FUNCTION_BLOCK FB_Mover EXTENDS CyclicBase IMPLEMENTS IMover, IDynamics
VAR
	axesEnable		: AxisPower(_axis);
	axesReset		: AxesReset(_axis);
	axesMoveTo 		: MoveMoverToPosition(_axis) := (Gap := 100.0);
	axesHalt 		: HaltMover(_axis);
	axesReadError : Tc2_MC2.MC_ReadAxisError;
	_axis 			: AXIS_REF;
	_identInGroup : INT;
	_trackLength : MC_LREAL;
	_targetPos : LREAL;
	_MoverErrorId : DWORD;
	_arrZones : ARRAY[1..4] OF DINT;
	_arrVelocities : ARRAY[1..4] OF mc_LREAL;
END_VAR

PROPERTY PUBLIC Acceleration : mc_lreal
GET
Acceleration := axesMoveTo.Acceleration;
END_GET
SET
axesMoveTo.Acceleration := Acceleration;
END_SET
END_PROPERTY

PROPERTY PUBLIC AxisRef : reference to AXIS_REF
GET
AxisRef REF= THIS^._axis;
END_GET
END_PROPERTY

METHOD PUBLIC  Cycle : BOOL
VAR_INPUT
END_VAR
axesMoveTo.Cycle();
axesHalt.Cycle();
axesReset.Cycle();
_axis.ReadStatus();
axesEnable.Cycle();
axesReadError(Axis := _axis, Enable := TRUE, AxisErrorID => _MoverErrorId);
END_METHOD

PROPERTY PUBLIC Deceleration : mc_lreal
GET
Deceleration := axesMoveTo.Deceleration;
END_GET
SET
axesMoveTo.Deceleration := Deceleration;
END_SET
END_PROPERTY

METHOD PUBLIC DisableAxis : BOOL
VAR_INPUT
END_VAR
DisableAxis := axesEnable.Disable();
END_METHOD

METHOD PUBLIC EnableAxis : BOOL
VAR_INPUT
END_VAR
EnableAxis := axesEnable.Enable();
END_METHOD

PROPERTY PUBLIC Gap : mc_lreal
GET
Gap := axesMoveTo.Gap;
END_GET
SET
axesMoveTo.Gap := Gap;
END_SET
END_PROPERTY

METHOD PUBLIC HaltAxis : BOOL
VAR_INPUT
END_VAR
IF NOT axesHalt.Busy THEN
	axesHalt.Execute();
	HaltAxis := TRUE;
	axesMoveTo.Abort();
END_IF
END_METHOD

METHOD PUBLIC HasCommand : BOOL
VAR_INPUT
END_VAR
HasCommand := axesMoveTo.Busy;
END_METHOD

METHOD hasError : BOOL
VAR_INPUT
END_VAR
hasError := _axis.Status.Error;
END_METHOD

PROPERTY PUBLIC IdentInGroup : int
GET
IdentInGroup := _identInGroup;
END_GET
SET
_identInGroup := IdentInGroup;
END_SET
END_PROPERTY

METHOD isAtPosition : BOOL
VAR_INPUT
	position : MC_LREAL;
END_VAR
IF position > 1 THEN
	IF _axis.NcToPlc.ModuloActPos < position + 1 AND _axis.NcToPlc.ModuloActPos > position - 1 THEN
		isAtPosition := TRUE;
	END_IF  
ELSE
	IF _axis.NcToPlc.ModuloActPos < position + 1 AND _axis.NcToPlc.ModuloActPos > 0.0  
		OR _axis.NcToPlc.ModuloActPos < _trackLength AND _axis.NcToPlc.ModuloActPos > _trackLength - 1 THEN
		isAtPosition := TRUE;
	END_IF
END_IF
END_METHOD

METHOD PUBLIC isDetected : BOOL
VAR_INPUT
END_VAR
IF _axis.NcToPlc.AxisId = 0 THEN
	RETURN;
END_IF
isDetected := true;
END_METHOD

METHOD isEnabled : BOOL
VAR_INPUT
END_VAR
isEnabled := not _axis.Status.Disabled;
END_METHOD

METHOD PUBLIC isPastPosition : BOOL
VAR_INPUT
	position : MC_LREAL;
END_VAR
IF position > 1 THEN
	IF _axis.NcToPlc.ModuloActPos > position THEN
		isPastPosition := TRUE;
	END_IF  
END_IF
END_METHOD

METHOD PUBLIC isStationary : BOOL
VAR_INPUT
END_VAR
isStationary := _axis.NcToPlc.SetVelo = 0;
END_METHOD

PROPERTY PUBLIC Jerk : mc_lreal
GET
Jerk := axesMoveTo.Jerk;
END_GET
SET
axesMoveTo.Jerk := Jerk;
END_SET
END_PROPERTY

METHOD PROTECTED ModuloToAbs : mc_lreal
VAR_INPUT
	moduloPositionDemand: MC_LREAL;
	_backwardsAllowed : BOOL;
END_VAR
//---------code to set actual position from modulo command----------------------
IF NOT _backwardsAllowed THEN
	//--------if you want to go forward-------------------------------------------------------------
	//---------if SetPos is greater than current actual then move to that position--------------------
	//---------else current position is greater, increase moduloturn count by 1 before set---------------
	IF moduloPositionDemand > _axis.NcToPlc.ModuloActPos THEN
		ModuloToAbs := (DINT_TO_LREAL(_Axis.NcToPlc.ModuloActTurns)*_trackLength) + moduloPositionDemand;
	ELSE
		ModuloToAbs := (DINT_TO_LREAL(_Axis.NcToPlc.ModuloActTurns + 1)*_trackLength) + moduloPositionDemand;
	END_IF
ELSE
	//--------if you want to go backwards--------------------------------
	//--------if setPos is less than current actual then move to that position---------------------
	//---------else current position is less, decrease moduloturn count by 1 before set------------
	IF moduloPositionDemand < _axis.NcToPlc.ModuloActPos THEN
		ModuloToAbs := (DINT_TO_LREAL(_Axis.NcToPlc.ModuloActTurns)*_trackLength) + moduloPositionDemand;
	ELSE
		ModuloToAbs := (DINT_TO_LREAL(_Axis.NcToPlc.ModuloActTurns-1)*_trackLength) + moduloPositionDemand;
	END_IF
END_IF
END_METHOD

PROPERTY MoverErrorId : dword
GET
MoverErrorId := _MoverErrorId;
END_GET
SET
_MoverErrorId := MoverErrorId;
END_SET
END_PROPERTY

METHOD PUBLIC MoveTo : BOOL
VAR_INPUT
	Position : MC_LREAL;
	Velocity : MC_LREAL;
	BackwardMove : BOOL;
END_VAR
IF NOT isAtPosition(position := Position) THEN
	IF NOT axesMoveTo.Busy THEN
		axesMoveTo.MoveTo(Position := ModuloToAbs(Position, BackwardMove), Velocity := Velocity);
		MoveTo := TRUE;
		_targetPos := Position;
	END_IF
END_IF
END_METHOD

METHOD PUBLIC ResetAxis : BOOL
VAR_INPUT
END_VAR
VAR
END_VAR
axesReset.Execute();
axesMoveTo.Abort();
axesHalt.Abort();
END_METHOD

PROPERTY PUBLIC TrackLength : MC_LREAL
GET
TrackLength := _trackLength;
END_GET
SET
_trackLength := TrackLength;
END_SET
END_PROPERTY

PROPERTY Zones : array[1..4] of dint
GET
Zones := _arrZones;
END_GET
SET
_arrZones := Zones;
END_SET
END_PROPERTY

PROPERTY ZoneVelocities : array[1..4] of mc_lreal
GET
ZoneVelocities := _arrVelocities;
END_GET
SET
_arrVelocities := ZoneVelocities;
END_SET
END_PROPERTY

END_FUNCTION_BLOCK

(* stored: Version 1.1.0.1, ProductVersion 3.1.4024.12
   POU FB_Mover: Id {8d73ea9c-992c-45cc-86ce-646b77b87654}, SpecialFunc None
   Folder Methods: Id {11c06f36-011b-43e0-ba96-46cd7b32bc9c}
   Folder Properties: Id {a74425e5-3b65-414c-b3c2-ebd17b6452b3}
   Property Acceleration: Id {189e8681-4788-4e2c-a142-1a297a08acd8}
   Get Get: Id {2a072cec-dc98-4e3e-832d-7b1661a2a48e}
   Set Set: Id {ac96b1c2-72ed-4693-b71f-9fbcd2a6afd7}
   Property AxisRef: Id {09529bdd-b0dc-4149-87fe-1e673dd7e409}
   Get Get: Id {8057bced-3b30-4db1-bed6-093c25080d45}
   Method Cycle: Id {df169178-ee0f-491e-a015-1bc9be6eb17c}
   Property Deceleration: Id {c85f3f81-4f88-4542-92dd-87b98693dee4}
   Get Get: Id {578458d3-d8f3-428d-9fc2-a6d51c86d4b3}
   Set Set: Id {b756c826-c655-4fcf-88a7-bb105c6d7b9b}
   Method DisableAxis: Id {c70711cc-2b37-46ae-851d-9b38023a0d20}
   Method EnableAxis: Id {b661d1e7-696c-4d63-afd0-3918405db14b}
   Property Gap: Id {e555cbf2-c13b-4254-9bb2-744e7edb7578}
   Get Get: Id {a0479bdd-653c-4687-93eb-073972457858}
   Set Set: Id {8af53078-5c57-4e61-9843-6d0cf8d12af4}
   Method HaltAxis: Id {fcdbac8a-7893-40e4-99e2-5063962a86e4}
   Method HasCommand: Id {87052920-e2d9-4076-9a13-adb664b2e231}
   Method hasError: Id {c0115f9f-d324-4748-af93-c56fdaaf010c}
   Property IdentInGroup: Id {ef5d4455-d34d-4ca1-b17f-13425cd154ed}
   Get Get: Id {de907afb-d6b6-48b4-8857-851ff7b7bba8}
   Set Set: Id {4b095c67-211b-468a-8be3-48d4ac28c572}
   Method isAtPosition: Id {2f15d1ba-ddfc-4b9e-afe4-5a0e456096bb}
   Method isDetected: Id {4d5c40c2-9705-45a9-9e7d-17e4126ba8ba}
   Method isEnabled: Id {5db97821-4f9e-4a12-8756-664c948ce8d4}
   Method isPastPosition: Id {9fa8306a-b12e-4f44-a97a-94fb24ba9f28}
   Method isStationary: Id {38624f60-08a0-42b1-ae6f-e7cfbf630206}
   Property Jerk: Id {08f26a51-2cac-4172-adfd-333cdfa23de5}
   Get Get: Id {b3f4bc4a-fc36-46a7-a0ff-605d9a2ddc0b}
   Set Set: Id {e967ae27-5c59-444d-a01e-9a7980e3667f}
   Method ModuloToAbs: Id {3e98c8eb-3ddf-4e09-8a71-47cbd2f60d1c}
   Property MoverErrorId: Id {9dd8a1e0-fec3-4fe1-b6c7-7672f776d3e1}
   Get Get: Id {5d87ebfd-264d-4297-a88a-3a51effeabaa}
   Set Set: Id {2d976bdd-4699-43a1-a341-b5a154776a7a}
   Method MoveTo: Id {22b20b94-6b3d-4a28-b255-aa56b1b14669}
   Method ResetAxis: Id {3034fc38-9b42-4179-8f04-b3d56b63ba9c}
   Property TrackLength: Id {17360115-9dc5-4ca9-8916-892bf20db53d}
   Get Get: Id {c5663a5c-fa26-4ec2-af50-b07c4b33da3f}
   Set Set: Id {a4b21aac-be54-4051-8d48-658c2585f98e}
   Property Zones: Id {c1269f03-c64a-4c39-99c0-152b4e2ef4a7}
   Get Get: Id {ec2f2417-7e7b-4e6b-8c00-7da02bf2a995}
   Set Set: Id {439816ee-60ba-41e6-9de0-9341cdae8b08}
   Property ZoneVelocities: Id {52ce116e-4240-4245-a327-1f542f2454ed}
   Get Get: Id {310e4d19-d444-4356-a27d-86c9ecf1e695}
   Set Set: Id {d19e7a94-d331-4553-92b6-b1de294924bf} *)
